SUBAPPLICATION Uebung_020c4_AX (* DigitalInput_I1 auf DigitalOutput_Q1; E_TON Einschaltverzögert; Zeit eingeben und speichern, INI *)
  (* Standard: 61499-2; Description: Copyright (c) 2023 Meisterschulen am Ostbahnhof This program and the accompanying materials are made available under the terms of the Eclipse Public License 2.0 which is available at https://www.eclipse.org/legal/epl-2.0/ SPDX-License-Identifier: EPL-2.0 *)
  (* Version 1.0, 2023-10-23, Franz Höpfinger, Meisterschulen am Ostbahnhof, initial API and implementation and/or initial documentation *)
  PACKAGE Uebungen;
  IMPORT Uebungen::const::NVS::NVS_Keys::KEY_I1_STORE;
  IMPORT Uebungen::const::NVS::NVS_Keys::SECTION_I1_STORE;
  IMPORT Uebungen::const::UT::DefaultPool_Numeric::InputNumber_I1_N;
  IMPORT logiBUS::io::DI::logiBUS_DI::Input_I1;
  IMPORT logiBUS::io::DQ::logiBUS_DO::Output_Q1;
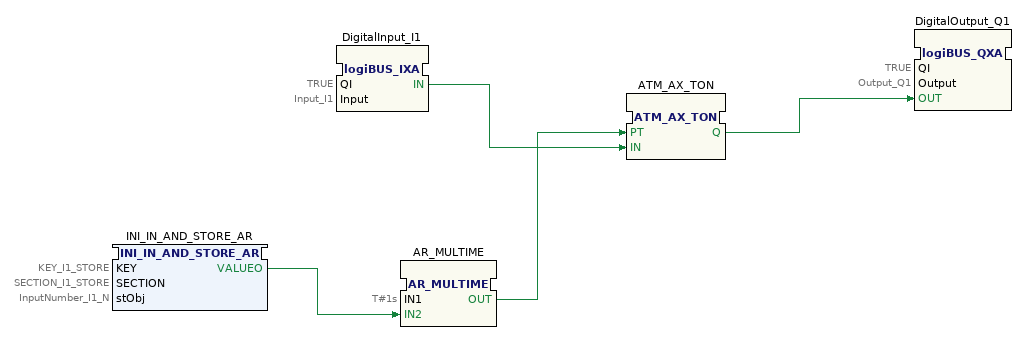
  FBS
    DigitalOutput_Q1 : logiBUS::io::DQ::logiBUS_QXA(QI := TRUE, Output := Output_Q1);
    DigitalInput_I1 : logiBUS::io::DI::logiBUS_IXA(QI := TRUE, Input := Input_I1);
    ATM_AX_TON : adapter::events::unidirectional::timers::ATM_AX_TON;
    AR_MULTIME : adapter::iec61131::arithmetic::AR_MULTIME(IN1 := T#1s);
  END_FBS
  SUBAPPS
    INI_IN_AND_STORE_AR : MyLib::sys::INI_IN_AND_STORE_AR(KEY := KEY_I1_STORE, SECTION := SECTION_I1_STORE, stObj := InputNumber_I1_N);
  END_SUBAPPS
  ADAPTER_CONNECTIONS
    AR_MULTIME.OUT TO ATM_AX_TON.PT;
    DigitalInput_I1.IN TO ATM_AX_TON.IN;
    ATM_AX_TON.Q TO DigitalOutput_Q1.OUT;
    INI_IN_AND_STORE_AR.VALUEO TO AR_MULTIME.IN2;
  END_CONNECTIONS
END_SUBAPPLICATION
